ABB RobotStudio station: soft.rsstn

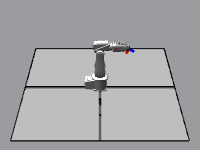
Station soft (saved by RobotStudio 6.8.8148.134)
Controller IRB_120_3kg_0.58m
  mechanical unit ROB_1: IRB120_3_58__01, 6 joints, base frame (0, 0, 0) mm
Layout (positions relative to the parent item):
  - IRB120_3_58__01 [mechanism, from Robots\IRB120_3_58_G_01.rslib] at (0, 0, 0) mm; joint values [0, 0, 0, 0, 0.5236, 0] (rad or m)
Targets, tools, work objects and paths stored in the station, written as RAPID:
! task T_ROB1
MODULE Module1
  PROC main()
    WaitTime 100;
  ENDPROC
ENDMODULE

! task T_ROB1
MODULE movement
  PROC Test13()
    WaitTime 100;
  ENDPROC
ENDMODULE

